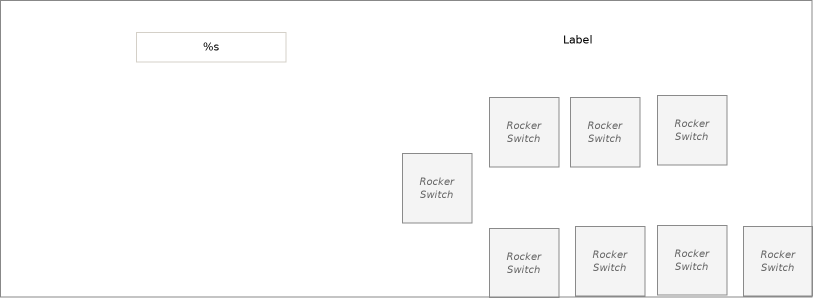
VISUALIZATION TAB_Simulation  // 813x298
    RockerSwitch (489,97 70x70), variable: MAIN.fbMachine.fbMPG.bX1, behaviour: TOGGLE, style: Switch-RockerSwitch-Blue
    RockerSwitch (570,97 70x70), variable: MAIN.fbMachine.fbMPG.bX10, behaviour: TOGGLE, style: Switch-RockerSwitch-Blue
    RockerSwitch (657,95 70x70), variable: MAIN.fbMachine.fbMPG.bX100, behaviour: TOGGLE, style: Switch-RockerSwitch-Blue
    RockerSwitch (402,153 70x70), behaviour: TOGGLE, style: Switch-RockerSwitch-Blue
    RockerSwitch (489,228 70x70), behaviour: TOGGLE, style: Switch-RockerSwitch-Blue
    RockerSwitch (575,226 70x70), behaviour: TOGGLE, style: Switch-RockerSwitch-Blue
    RockerSwitch (657,225 70x70), behaviour: TOGGLE, style: Switch-RockerSwitch-Blue
    RockerSwitch (743,226 70x70), behaviour: TOGGLE, style: Switch-RockerSwitch-Blue
    Label (503,25 150x30), "Label"
    Textfield (136,32 150x30), "%s", text variable: MAIN.fbMachine.fbVisu.sDisplayText_MPG
END_VISUALIZATION

(* stored: Version 1.1.0.1, ProductVersion 3.1.4024.11
   Visu TAB_Simulation: Id {d089075f-220a-4eec-8047-c343388baefb} *)
